// TIA Portal V19 export
TYPE "LEXCHANGETRAY_typeMaterialMonitor"
// stored: Access Published
   STRUCT
      cells : "LEXCHANGETRAY_typeCellsMonitor";   // 托盘状态
      tray { S7_SetPoint := 'True'} : "LEXCHANGETRAY_typeTrayMonitor";
   END_STRUCT;
END_TYPE
